// TIA Portal V17 export
// export: Created 2024-09-02T12:50:33.4987645Z, ExportSetting WithDefaults, DisplayName Totally Integrated Automation Portal, DisplayVersion V17, DisplayName TIA Portal Openness, DisplayVersion V17, DisplayName TIA Portal Version Control Interface, DisplayVersion V17, DisplayName STEP 7 Professional, DisplayVersion V17, DisplayName STEP 7 Safety, DisplayVersion V17, DisplayName WinCC Professional, DisplayVersion V17
TYPE "TypeMobyBefehleBIS"
// stored: IsFailsafeCompliant false
   STRUCT
      Sequenz { S7_SetPoint := 'True'} : "TypeMobySequenzBIS";
      DatenPuffer { S7_SetPoint := 'True'} : "TypeMobyDatenPufferBIS";
      GroessePuffer : UDInt;
   END_STRUCT;
END_TYPE
